Universal Robots PolyScope program: translation_sample_servoj_torque.urp

Program translation_sample_servoj_torque (installation=default directory=/programs/usbdisk createdIn=3.2.19275.0 lastSavedIn=5.12.0.1101482 robotSerialNumber=20225501047)
Calibrated DH parameters: a=[0.000165, -0.414236, -0.366713, 0.000028, 0.000067, 0]; d=[0.162801, -57.2398, 32.079015, 25.294245, 0.099708, 0.099569]; alpha=[1.570474, 0.001669, 0.005558, 1.570315, -1.568415, 0]; deltaTheta=[0, -0.226697, 6.145588, 0.364296, 0.000001, 0]
BeforeStart
  joints := get_actual_joint_positions()
  cdio := integer_to_binary_list(0)
  Script: write_output_boolean_register(0, False )
  Wait Sleep waitTime=0.01
  Script: popup("Registers reset, run PC code and then click Continue",title="Hi Daniel",blocking= True )
  mode := 0
Robot Program (runOnlyOnce=false)
  Script: write_output_boolean_register(0, True )
  Script: sync()
  Loop While (checkContinuously=false) expression=mode<3
    Loop While (checkContinuously=false) expression=mode≟1
      Set ExpressionOutput pin=config_out[0]; expression=cdio[0]
      Set ExpressionOutput pin=config_out[1]; expression=cdio[1]
      Set ExpressionOutput pin=config_out[2]; expression=cdio[2]
      MoveJ speed 60 deg/s, acceleration 80 deg/s^2 (useActiveTCP=true) feature=Base
        Waypoint Waypoint (Variable): variable(name=joints)
      Script: write_output_boolean_register(0, False )
      Script: sync()
    Loop While (checkContinuously=false) expression=mode≟2
      Set ExpressionOutput pin=config_out[2]; expression=cdio[2]
      Set ExpressionOutput pin=config_out[0]; expression=cdio[0]
      Set ExpressionOutput pin=config_out[1]; expression=cdio[1]
      Script: servoj(joints, 0, 0, 0.002, 0.03, 2000)
    Loop While (checkContinuously=false) expression=mode≟3
      Set ExpressionOutput pin=config_out[0]; expression=False
      Set ExpressionOutput pin=config_out[1]; expression=False
      Set ExpressionOutput pin=config_out[2]; expression=False
      Halt
  Script: sync()
Thread Thread_1 (runOnlyOnce=false)
  tmp := get_actual_joint_positions()
  cdio_tmp := 0
  Loop Forever
    Script file /programs/pose_register.script
      | tmp[0]=read_input_float_register(0)
      | tmp[1]=read_input_float_register(1)
      | tmp[2]=read_input_float_register(2)
      | tmp[3]=read_input_float_register(3)
      | tmp[4]=read_input_float_register(4)
      | tmp[5]=read_input_float_register(5)
      | cdio_tmp=read_input_integer_register(1)
    joints := [tmp[0],tmp[1],tmp[2],tmp[3],tmp[4],tmp[5]]
    cdio := integer_to_binary_list(cdio_tmp)
    Script: sync()
    mode := read_input_integer_register(0)
    Script: sync()
